{attribute 'qualified_only'}
VAR_GLOBAL CONSTANT
    DICTIONARY_UPPER_BOUND : INT := 4;
END_VAR

(* stored: Version 1.1.0.1, ProductVersion 3.1.4024.12
   GVL GVL: Id {bbb8674d-7996-4211-9872-cb0b304073a4} *)
